Omron CX-Programmer project NewProject (CX-Programmer 9.73)

# PLC NewPLC1: CP1E E30

## Global symbols (name address type ; comment)
0.01 BOOL  ; suis 1
0.02 BOOL  ; suis2
0.03 BOOL  ; suis lamp
100.00 BOOL  ; motor 1
100.01 BOOL  ; motor 2
100.03 BOOL  ; lamp

## Program NewProgram1 (cyclic task 0)

### Section Section1

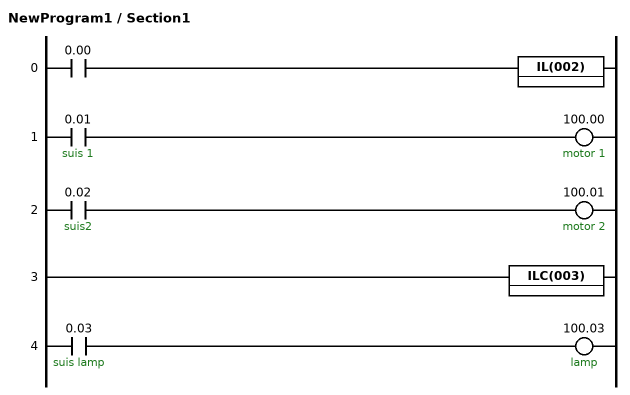
; rung 0
LD 0.00
IL(002)
; rung 1
LD 0.01  ; suis 1
OUT 100.00  ; motor 1
; rung 2
LD 0.02  ; suis2
OUT 100.01  ; motor 2
; rung 3
ILC(003)
; rung 4
LD 0.03  ; suis lamp
OUT 100.03  ; lamp

### Section END
; rung 0
END(001)